TYPE ST_FloorOne :
STRUCT
	
	{attribute 'iot.NestedStructIcon' := 'Lightbulb'}
	{attribute 'iot.DisplayName' := 'Light Widgets'}
	stLights		: ST_Lighting;
	
	{attribute 'iot.NestedStructIcon' := 'Room'}
	{attribute 'iot.DisplayName' := 'Confrence Room'}
	stF1RoomOne		: ST_F1RoomOne;

END_STRUCT
END_TYPE

(* stored: Version 1.1.0.1, ProductVersion 3.1.4024.12
   DUT ST_FloorOne: Id {c02cf3b7-43db-45f9-9ccd-8fbd2414f672} *)
